INTERFACE I_BinaryDevice EXTENDS I_HMIBase

END_INTERFACE

(* stored: Version 1.1.0.1
   Itf I_BinaryDevice: Id {23f75292-a9cd-4826-8fd6-29dab4d849ea} *)
